// TIA Portal V20 export
// export: Created 2026-04-11T06:02:30.8027386Z, ExportSetting WithDefaults, DisplayName Totally Integrated Automation Portal, DisplayVersion V20, DisplayName TIA Portal Openness, DisplayVersion V20, DisplayName TIA Portal Version Control Interface, DisplayVersion V20, DisplayName STEP 7 Professional, DisplayVersion V20, DisplayName STEP 7 Safety, DisplayVersion V20, DisplayName WinCC Basic/Comfort/Advanced, DisplayVersion V20, DisplayName WinCC Unified, DisplayVersion V20
TYPE "udtQueue"
// stored: IsFailsafeCompliant false
   STRUCT
      bEnabled { ExternalWritable := 'False'} : Bool;   // Queue is enabled for dequeuing
      iQueuedCount { ExternalWritable := 'False'} : Int;   // Number of items in the queue
      iSelectedItem { ExternalWritable := 'False'} : Int;   // Currently selected queue item
      Item { ExternalWritable := 'False'; S7_SetPoint := 'True'} : Array[1.."FIFO.iQueueSize"] of "udtQueueItem";   // The queue
   END_STRUCT;
END_TYPE
